TYPE RecipeStep :
STRUCT
	sRecipe : STRING(81);
	iRecipe : ARRAY[1..5] OF INT; //Reactor Condition
	rRecipe : ARRAY[1..GVL_IO.nNumController] OF REAL; //MFC, Furnace Temp
	dRecipe : DWORD; //Valve Data
END_STRUCT
END_TYPE

(* stored: Version 1.1.0.1
   DUT RecipeStep: Id {c67477fa-59d3-43d0-9335-dff43a63186e} *)
